FUNCTION_BLOCK KnownExamplesTest EXTENDS TcUnit_Zeugwerk.FB_TestSuite

example01();
example02();
example03();
example04();
example05();
example06();
example07();
example08();
example09();
example10();
example11();
example12();
example13();
example14();
example15();
example16();
example17();
example18();
example19();
example20();
example21();
example22();
example23();
example24();
example25();
example26();
example27();
example28();
example29();
example30();
example31();
example32();
example33();
example34();
example35();
example36();
example37();

METHOD example01
VAR_INST
  otg : Struckig.Otg(0.005, 3) := (
  
    Synchronization := SynchronizationType.None,        
    MaxVelocity :=         [ 1.0, 1.0, 1.0 ],
    MaxAcceleration :=     [ 1.0, 1.0, 1.0 ],
    MaxJerk :=             [ 1.0, 1.0, 1.0 ],
    CurrentPosition :=     [ 0.0, 0.0, 0.0 ],
    CurrentVelocity :=     [ 0.0, 0.0, 0.0 ],
    CurrentAcceleration := [ 0.0, 0.0, 0.0 ],
    TargetPosition :=      [ 0.0, 0.0, 0.0 ],
    TargetVelocity :=      [ 0.0, 0.0, 0.0 ],
    TargetAcceleration :=  [ 0.0, 0.0, 0.0 ]
  );
  
END_VAR
TEST('Example-01');

otg();
AssertEquals_LREAL(Expected := 0.0,
             Actual := CheckCalculation(otg),
             DELTA := 1E-8,
             Message := '');
 
TEST_FINISHED();
END_METHOD

METHOD example02
VAR_INST
  otg : Struckig.Otg(0.005, 3) := (
  
    Synchronization := SynchronizationType.None,        
    MaxVelocity :=         [ 1.0, 1.0, 1.0 ],
    MaxAcceleration :=     [ 1.0, 1.0, 1.0 ],
    MaxJerk :=             [ 1.0, 1.0, 1.0 ],
    CurrentPosition :=     [ 0.0, 0.0, 0.0 ],
    CurrentVelocity :=     [ 0.0, 0.0, 0.0 ],
    CurrentAcceleration := [ 0.0, 0.0, 0.0 ],
    TargetPosition :=      [ 0.0, 1E-17, -1E-17 ],
    TargetVelocity :=      [ 0.0, 0.0, 0.0 ],
    TargetAcceleration :=  [ 0.0, 0.0, 0.0 ]
  );
    
END_VAR
TEST('Example-02');

otg();
AssertEquals_LREAL(Expected := 1E-18,
             Actual := CheckCalculation(otg),
             Delta := 1E-8,
             Message := '');
 
TEST_FINISHED();
END_METHOD

METHOD example03
VAR_INST
  otg : Struckig.Otg(0.005, 3) := (
  
    Synchronization := SynchronizationType.None,        
    MaxVelocity :=         [ 1.0, 1.0, 1.0 ],
    MaxAcceleration :=     [ 1.0, 1.0, 1.0 ],
    MaxJerk :=             [ 1.0, 1.0, 1.0 ],
    CurrentPosition :=     [ 0.0, 1E-17, -1E-17 ],
    CurrentVelocity :=     [ 0.0, 0.0, 0.0 ],
    CurrentAcceleration := [ 0.0, 0.0, 0.0 ],
    TargetPosition :=      [ 1.0, 1.0, 1.0 ],
    TargetVelocity :=      [ 0.0, 0.0, 0.0 ],
    TargetAcceleration :=  [ 0.0, 0.0, 0.0 ]
  );
  
  
END_VAR
TEST('Example-03');

otg();
AssertEquals_LREAL(Expected := 3.1748021039,
             Actual := CheckCalculation(otg),
             DELTA := 1E-8,
             Message := '');
 
TEST_FINISHED();
END_METHOD

METHOD example04
VAR_INST
  otg : Struckig.Otg(0.005, 3) := (
  
    Synchronization := SynchronizationType.None,        
    MaxVelocity :=         [ 1.0, 1.0, 1.0 ],
    MaxAcceleration :=     [ 1.0, 1.0, 1.0 ],
    MaxJerk :=             [ 2.0, 2.0, 2.0 ],
    CurrentPosition :=     [ 0.0, 0.0, 0.0 ],
    CurrentVelocity :=     [ 0.0, 0.0, 0.0 ],
    CurrentAcceleration := [ 0.0, 0.0, 0.0 ],
    TargetPosition :=      [ 1.0, 1.0, 1.0 ],
    TargetVelocity :=      [ 0.0, 0.0, 0.0 ],
    TargetAcceleration :=  [ 0.0, 0.0, 0.0 ]
  );
  
  
END_VAR
TEST('Example-04');

otg();
AssertEquals_LREAL(Expected := 2.5615528128,
             Actual := CheckCalculation(otg),
             DELTA := 1E-8,
             Message := '');
 
TEST_FINISHED();
END_METHOD

METHOD example05
VAR_INST
  otg : Struckig.Otg(0.005, 3) := (
  
    Synchronization := SynchronizationType.None,        
    MaxVelocity :=         [ 0.6, 0.6, 0.6 ],
    MaxAcceleration :=     [ 1.0, 1.0, 1.0 ],
    MaxJerk :=             [ 2.0, 2.0, 2.0 ],
    CurrentPosition :=     [ 0.0, 0.0, 0.0 ],
    CurrentVelocity :=     [ 0.0, 0.0, 0.0 ],
    CurrentAcceleration := [ 0.0, 0.0, 0.0 ],
    TargetPosition :=      [ 1.0, 1.0, 1.0 ],
    TargetVelocity :=      [ 0.0, 0.0, 0.0 ],
    TargetAcceleration :=  [ 0.0, 0.0, 0.0 ]
  );
  
  
END_VAR
TEST('Example-05');

otg();
AssertEquals_LREAL(Expected := 2.7666666667,
             Actual := CheckCalculation(otg),
             DELTA := 1E-8,
             Message := '');
 
TEST_FINISHED();
END_METHOD

METHOD example06
VAR_INST
  otg : Struckig.Otg(0.005, 3) := (
  
    Synchronization := SynchronizationType.None,        
    MaxVelocity :=         [ 0.4, 0.4, 0.4 ],
    MaxAcceleration :=     [ 1.0, 1.0, 1.0 ],
    MaxJerk :=             [ 2.0, 2.0, 2.0 ],
    CurrentPosition :=     [ 0.0, 0.0, 0.0 ],
    CurrentVelocity :=     [ 0.0, 0.0, 0.0 ],
    CurrentAcceleration := [ 0.0, 0.0, 0.0 ],
    TargetPosition :=      [ 1.0, 1.0, 1.0 ],
    TargetVelocity :=      [ 0.0, 0.0, 0.0 ],
    TargetAcceleration :=  [ 0.0, 0.0, 0.0 ]
  );
  	
END_VAR
TEST('Example-06');

otg();
AssertEquals_LREAL(Expected := 3.394427191,
             Actual := CheckCalculation(otg),
             DELTA := 1E-8,
             Message := '');
 
TEST_FINISHED();
END_METHOD

METHOD example07
VAR_INST
  otg : Struckig.Otg(0.005, 3) := (
  
    Synchronization := SynchronizationType.None,        
    MaxVelocity :=         [ 1.0, 1.0, 1.0 ],
    MaxAcceleration :=     [ 1.0, 1.0, 1.0 ],
    MaxJerk :=             [ 2.0, 2.0, 2.0 ],
    CurrentPosition :=     [ 0.0, 0.0, 0.0 ],
    CurrentVelocity :=     [ 0.3, 0.3, 0.3 ],
    CurrentAcceleration := [ 0.0, 0.0, 0.0 ],
    TargetPosition :=      [ 1.0, 1.0, 1.0 ],
    TargetVelocity :=      [ 0.0, 0.0, 0.0 ],
    TargetAcceleration :=  [ 0.0, 0.0, 0.0 ]
  );
  
  
END_VAR
TEST('Example-07');

otg();
AssertEquals_LREAL(Expected := 2.2319602829,
             Actual := CheckCalculation(otg),
             DELTA := 1E-8,
             Message := '');
 
TEST_FINISHED();
END_METHOD

METHOD example08
VAR_INST
  otg : Struckig.Otg(0.005, 3) := (
  
    Synchronization := SynchronizationType.None,        
    MaxVelocity :=         [ 0.6, 0.6, 0.6 ],
    MaxAcceleration :=     [ 1.0, 1.0, 1.0 ],
    MaxJerk :=             [ 2.0, 2.0, 2.0 ],
    CurrentPosition :=     [ 0.0, 0.0, 0.0 ],
    CurrentVelocity :=     [ 0.3, 0.3, 0.3 ],
    CurrentAcceleration := [ 0.0, 0.0, 0.0 ],
    TargetPosition :=      [ 1.0, 1.0, 1.0 ],
    TargetVelocity :=      [ 0.0, 0.0, 0.0 ],
    TargetAcceleration :=  [ 0.0, 0.0, 0.0 ]
  );
  
  
END_VAR
TEST('Example-08');

otg();
AssertEquals_LREAL(Expected := 2.410315834,
             Actual := CheckCalculation(otg),
             DELTA := 1E-8,
             Message := '');
 
TEST_FINISHED();
END_METHOD

METHOD example09
VAR_INST
  otg : Struckig.Otg(0.005, 3) := (
  
    Synchronization := SynchronizationType.None,        
    MaxVelocity :=         [ 0.6, 0.6, 0.6 ],
    MaxAcceleration :=     [ 1.0, 1.0, 1.0 ],
    MaxJerk :=             [ 2.0, 2.0, 2.0 ],
    CurrentPosition :=     [ 0.0, 0.0, 0.0 ],
    CurrentVelocity :=     [ 0.0, 0.0, 0.0 ],
    CurrentAcceleration := [ 0.0, 0.0, 0.0 ],
    TargetPosition :=      [ -1.0, -1.0, -1.0 ],
    TargetVelocity :=      [ 0.0, 0.0, 0.0 ],
    TargetAcceleration :=  [ 0.0, 0.0, 0.0 ]
  );
  
  
END_VAR
TEST('Example-09');

otg();
AssertEquals_LREAL(Expected := 2.7666666667,
             Actual := CheckCalculation(otg),
             DELTA := 1E-8,
             Message := '');
 
TEST_FINISHED();
END_METHOD

METHOD example10
VAR_INST
  otg : Struckig.Otg(0.005, 3) := (
  
    Synchronization := SynchronizationType.None,        
    MaxVelocity :=         [ 10.0, 10.0, 10.0 ],
    MaxAcceleration :=     [ 10.0, 10.0, 10.0 ],
    MaxJerk :=             [ 2.0, 2.0, 2.0 ],
    CurrentPosition :=     [ 0.0, 0.0, 0.0 ],
    CurrentVelocity :=     [ 0.2, 0.2, 0.2 ],
    CurrentAcceleration := [ 0.0, 0.0, 0.0 ],
    TargetPosition :=      [ -1.0, -1.0, -1.0 ],
    TargetVelocity :=      [ 0.0, 0.0, 0.0 ],
    TargetAcceleration :=  [ 0.0, 0.0, 0.0 ]
  );
  
END_VAR
TEST('Example-10');

otg();
AssertEquals_LREAL(Expected := 2.7338531701,
             Actual := CheckCalculation(otg),
             DELTA := 1E-8,
             Message := '');
 
TEST_FINISHED();
END_METHOD

METHOD example11
VAR_INST
  otg : Struckig.Otg(0.005, 3) := (
  
    Synchronization := SynchronizationType.None,        
    MaxVelocity :=         [ 0.4, 0.4, 0.4 ],
    MaxAcceleration :=     [ 1.0, 1.0, 1.0 ],
    MaxJerk :=             [ 2.0, 2.0, 2.0 ],
    CurrentPosition :=     [ -1.0, -1.0, -1.0 ],
    CurrentVelocity :=     [ 0.2, 0.2, 0.2 ],
    CurrentAcceleration := [ 0.0, 0.0, 0.0 ],
    TargetPosition :=      [ 1.0, 1.0, 1.0 ],
    TargetVelocity :=      [ 0.0, 0.0, 0.0 ],
    TargetAcceleration :=  [ 0.0, 0.0, 0.0 ]
  );
  
  
END_VAR
TEST('Example-11');

otg();
AssertEquals_LREAL(Expected := 5.6053274785,
             Actual := CheckCalculation(otg),
             DELTA := 1E-8,
             Message := '');
 
TEST_FINISHED();
END_METHOD

METHOD example12
VAR_INST
  otg : Struckig.Otg(0.005, 3) := (
  
    Synchronization := SynchronizationType.None,        
    MaxVelocity :=         [ 3.0, 3.0, 3.0 ],
    MaxAcceleration :=     [ 0.5, 0.5, 0.5 ],
    MaxJerk :=             [ 0.2, 0.2, 0.2 ],
    CurrentPosition :=     [ 0.3888899206957 - 10E-14, 0.0, 0.0 ],
    CurrentVelocity :=     [ 0.2231429352410215, 0.0, 0.0 ],
    CurrentAcceleration := [ -0.2987593916455, 0.0, 0.0 ],
    TargetPosition :=      [ 0.5, 0.0, 0.0 ],
    TargetVelocity :=      [ 0.0, 0.0, 0.0 ],
    TargetAcceleration :=  [ 0.0, 0.0, 0.0 ]
  );
  
END_VAR
TEST('Example-12');

otg();
AssertEquals_LREAL(Expected := 1.493796958,
             Actual := CheckCalculation(otg),
             DELTA := 1E-8,
             Message := '');
 
TEST_FINISHED();
END_METHOD

METHOD example13
VAR_INST
  otg : Struckig.Otg(0.005, 3) := (
  
    Synchronization := SynchronizationType.None,        
    MaxVelocity :=         [ 12.9892953062198, 3.74169932927481, 1.42398447457303 ],
    MaxAcceleration :=     [ 4.2162106624246, 10.2906731766853, 2.1869079548297 ],
    MaxJerk :=             [ 8.03496976453435, 0.200684346397485 - 1.0E-14, 0.0848503482861296 ],
    CurrentPosition :=     [ -5.54640573838539, -2.34195463203842, 5.10070661762967 ],
    CurrentVelocity :=     [ 0.824843228617216, -1.03863337183304, -0.749451523227729 ],
    CurrentAcceleration := [ -0.119403564898501, 0.923861820607788, 3.04022341347259 ],
    TargetPosition :=      [ -1.58293112753888, 0.383405919465141, 5.79349604610299 ],
    TargetVelocity :=      [ -1.59453676324393, 0.0, -0.0693173526513803 ],
    TargetAcceleration :=  [ -0.664429703711622, 0.0, 0.0 ]
  );
  
  
END_VAR
TEST('Example-13');

otg();
AssertEquals_LREAL(Expected := 1921.0797627836,
             Actual := CheckCalculation(otg),
             DELTA := 1E-8,
             Message := '');
 
TEST_FINISHED();
END_METHOD

METHOD example14
VAR_INST
  otg : Struckig.Otg(0.005, 3) := (
  
    Synchronization := SynchronizationType.None,        
    MaxVelocity :=         [ 8.65978706670502, 5.94921088330542, 10.7652253566829 ],
    MaxAcceleration :=     [ 3.40137210377608, 4.04166318018487, 10.8617860610581 ],
    MaxJerk :=             [ 10.9542353113865, 3.11056302676629, 0.798055744482636 + 9E-12 ],
    CurrentPosition :=     [ -6.49539540831446, 6.14883133273172, -2.02636240900911 ],
    CurrentVelocity :=     [ -1.14327601654428, 0.00991019970085593, -1.00932863927626 ],
    CurrentAcceleration := [ -1.73501068960131, -0.584885092422228, 0 ],
    TargetPosition :=      [ 4.4676187540058, 2.93367894961155, -0.646008452514058 ],
    TargetVelocity :=      [ -0.544559915133859, 0.298517792372943, 1.6058847848484 ],
    TargetAcceleration :=  [ -1.31832055647831, 0, 0 ]
  );
  
  
END_VAR
TEST('Example-14');

otg();
AssertEquals_LREAL(Expected := 4.6277455678,
             Actual := CheckCalculation(otg),
             DELTA := 1E-8,
             Message := '');
 
TEST_FINISHED();
END_METHOD

METHOD example15
VAR_INST
  otg : Struckig.Otg(0.005, 3) := (
  
    Synchronization := SynchronizationType.TimeSync,        // TODO: there seems to be a bug here, if set to None, the reported duration is <3s
    MaxVelocity :=         [ 7.97399137456765, 2.68591430972239, 9.54987666746364 ],
    MaxAcceleration :=     [ 5.44679859206862, 7.61752909348119, 0.473482772614085 ],
    MaxJerk :=             [ 7.88958080921515, 5.26855927512131, 0.764061581326592 - 1E-14 ],
    CurrentPosition :=     [ 7.06378251402596, -2.4834697862831, -0.843847405371359 ],
    CurrentVelocity :=     [ 0.436985859305842, 0.0708113515655622, -0.751266816040307 ],
    CurrentAcceleration := [ -0.80835350359544, 0, -0.355284934641626 ],
    TargetPosition :=      [ 4.40606827118048, -2.84629921001043, -2.91829890043522 ],
    TargetVelocity :=      [ 0.555084596169823, 0, -1.24631524923535 ],
    TargetAcceleration :=  [ 0.463000173872542, 0, 0 ]
  );
  
  
END_VAR
TEST('Example-15');

otg();
AssertEquals_LREAL(Expected := 8.8739464323,
             Actual := CheckCalculation(otg),
             DELTA := 1E-8,
             Message := '');
 
TEST_FINISHED();
END_METHOD

METHOD example16
VAR_INST
  otg : Struckig.Otg(0.005, 3) := (
  
    Synchronization := SynchronizationType.None,        
    MaxVelocity :=         [ 0.1241065584614779, 1, 1 ],
    MaxAcceleration :=     [ 1.808598147153279, 1, 1 ],
    MaxJerk :=             [ 2.516849090900998 - 3E-15, 1, 1 ],
    CurrentPosition :=     [ -7.962737259350095, 0, 0 ],
    CurrentVelocity :=     [ -0.8844863500141733, 0, 0 ],
    CurrentAcceleration := [ 2.252932547031004, 0, 0 ],
    TargetPosition :=      [ -3.547368989678775, 0, 0 ],
    TargetVelocity :=      [ 0, 0, 0 ],
    TargetAcceleration :=  [ 0.217242176687843, 0, 0 ]
  );
  
  
END_VAR
TEST('Example-16');

otg();
AssertEquals_LREAL(Expected := 38.3409477609,
             Actual := CheckCalculation(otg),
             DELTA := 1E-8,
             Message := '');
 
TEST_FINISHED();
END_METHOD

METHOD example17
VAR_INST
  otg : Struckig.Otg(0.005, 3) := (
  
    Synchronization := SynchronizationType.None,    
    MaxVelocity :=         [ 1.863775561344568, 0.4357836109021987, 6.260907804906162 ],
    MaxAcceleration :=     [ 9.49223908896113, 9.002562577262177, 1.119142029086944 ],
    MaxJerk :=             [ 8.689575453772798, 0.09322235504216797, 0.1594452521517275 + 3E-15 ],
    CurrentPosition :=     [ -4.180150148354134, 1.030371049895473, -2.660154279239869 ],
    CurrentVelocity :=     [ 1.673805463302308, -1.435796222257198, 0.9711306630275642 ],
    CurrentAcceleration := [ 1.412175048500792, 1.892262449040863, -1.128847905860926 ],
    TargetPosition :=      [ 2.079913937916431, 1.839862681333277, 2.341421542126605 ],
    TargetVelocity :=      [ 0.7537566830764975, 0, 0.02507782261105568 ],
    TargetAcceleration :=  [ -0.8610296259045267, -0.07876324073516261, 0 ]
  );
  
  
END_VAR
TEST('Example-17');

otg();
AssertEquals_LREAL(Expected := 1135.0135089249,
             Actual := CheckCalculation(otg),
             DELTA := 1E-8,
             Message := '');
 
TEST_FINISHED();
END_METHOD

METHOD example18
VAR_INST
  otg : Struckig.Otg(0.005, 3) := (
  
    Synchronization := SynchronizationType.None,
    MaxVelocity :=         [ 6.144314006624488, 2.93258338415229, 0.1820021269527196 ],
    MaxAcceleration :=     [ 5.199401036221791, 1.848176490768948, 11.11168017805234 ],
    MaxJerk :=             [ 9.940940357283978, 10.46997753899755, 0.08166297169205029 ],
    CurrentPosition :=     [ -4.490717417930574, 3.467236624628543, -0.7545929089757601 ],
    CurrentVelocity :=     [ 0.1839756723363622, -0.4356283320280516, 0.7490399525818022 ],
    CurrentAcceleration := [ -1.057769973808928, 0, -2.368645439140517 ],
    TargetPosition :=      [ -4.928244836531066, -4.821780824003112, -8.20567952461017 ],
    TargetVelocity :=      [ 0.1097319156272965, -0.9272874846270881, 0 ],
    TargetAcceleration :=  [ 0.03089046366221739, -0.9744054582899561, 0 ]
  );
  
  
END_VAR
TEST('Example-18');

otg();
AssertEquals_LREAL(Expected := 7295.4375633935,
             Actual := CheckCalculation(otg),
             DELTA := 1E-8,
             Message := '');
 
TEST_FINISHED();
END_METHOD

METHOD example19
VAR_INST
  otg : Struckig.Otg(0.005, 3) := (
  
    Synchronization := SynchronizationType.None,
    MaxVelocity :=         [ 1, 1, 1 ],
    MaxAcceleration :=     [ 7, 7, 7 ],
    MaxJerk :=             [ 1000, 1000, 1000 ],
    CurrentPosition :=     [ 0.01073568005271233, -0.7002627264230739, 0 ],
    CurrentVelocity :=     [ 0.05656281587106524, 1.011281770884991, 0 ],
    CurrentAcceleration := [ -5.348847133445708, -3.400994300842285, 0 ],
    TargetPosition :=      [ 0.0698, 0.6283, 0 ],
    TargetVelocity :=      [ 0, 0, 0 ],
    TargetAcceleration :=  [ 0, 0, 0 ]
  );
  
  
END_VAR
TEST('Example-19');

otg();
AssertEquals_LREAL(Expected := 1.403613276,
             Actual := CheckCalculation(otg),
             DELTA := 1E-3,
             Message := '');
 
TEST_FINISHED();
END_METHOD

METHOD example20
VAR_INST
  otg : Struckig.Otg(0.005, 3) := (
  
    Synchronization := SynchronizationType.None,
    MaxVelocity :=         [ 1, 1, 1 ],
    MaxAcceleration :=     [ 0.5, 0.5, 0.5 ],
    MaxJerk :=             [ 1, 1, 1 ],
    CurrentPosition :=     [ 0.0001215, 0, 0 ],
    CurrentVelocity :=     [ 0.00405, 0, 0 ],
    CurrentAcceleration := [ 0.09, 0, 0 ],
    TargetPosition :=      [ 0.1421083333333333087, 0, 0 ],
    TargetVelocity :=      [ 0.37, 0, 0 ],
    TargetAcceleration :=  [ 0.5, 0, 0 ]
  );
  
  
END_VAR
TEST('Example-20');

otg();
AssertEquals_LREAL(Expected := 0.9,
             Actual := CheckCalculation(otg),
             DELTA := 1E-8,
             Message := '');
 
TEST_FINISHED();
END_METHOD

METHOD example21
VAR_INST
  otg : Struckig.Otg(0.005, 3) := (
  
    Synchronization := SynchronizationType.None,
    MaxVelocity :=         [ 1800, 18000, 180000 ],
    MaxAcceleration :=     [ 20000, 200000, 2000000 ],
    MaxJerk :=             [ 200000, 2000000, 20000000 ],
    CurrentPosition :=     [ 0, 0, 0 ],
    CurrentVelocity :=     [ 0, 0, 0 ],
    CurrentAcceleration := [ 0, 0, 0 ],
    TargetPosition :=      [ 400, 4000, 40000 ],
    TargetVelocity :=      [ 0, 0, 0 ],
    TargetAcceleration :=  [ 0, 0, 0 ]
  );
  
  
END_VAR
TEST('Example-21');

otg();
AssertEquals_LREAL(Expected := 0.4119588818,
             Actual := CheckCalculation(otg),
             DELTA := 1E-8,
             Message := '');
 
TEST_FINISHED();
END_METHOD

METHOD example22
VAR_INST
  otg : Struckig.Otg(0.005, 3) := (
  
    Synchronization := SynchronizationType.None,
    MaxVelocity :=         [ 0.8500000000000001, 0.8500000000000001, 0.8500000000000001 ],
    MaxAcceleration :=     [ 4.25, 4.25, 4.25 ],
    MaxJerk :=             [ 85.00000000000001, 85.00000000000001, 85.00000000000001 ],
    CurrentPosition :=     [ -0.05598571695553641, -0.534847776106059, 0.0978130731424748 ],
    CurrentVelocity :=     [ -0.03425673149926184, -0.8169926404190487, -0.004506245841081729 ],
    CurrentAcceleration := [ -2.720000000000001, 1.440254448401435, 0 ],
    TargetPosition :=      [ -0.0534691276550293, -0.6224863891601563, 0.09690575408935546 ],
    TargetVelocity :=      [ 0, 0, 0 ],
    TargetAcceleration :=  [ 0, 0, 0 ]
  );
  
  
END_VAR
TEST('Example-22');

otg();
AssertEquals_LREAL(Expected := 0.2281604414,
             Actual := CheckCalculation(otg),
             DELTA := 1E-8,
             Message := '');
 
TEST_FINISHED();
END_METHOD

METHOD example23
VAR_INST
  otg : Struckig.Otg(0.005, 3) := (
  
    Synchronization := SynchronizationType.None,
    MaxVelocity :=         [ 1.0, 1.0, 10.01369296498101 ],
    MaxAcceleration :=     [ 1.0, 1.0, 14.72621077848741 ],
    MaxJerk :=             [ 1.0, 1.0, 7.770133554060553 ],
    CurrentPosition :=     [ 0.0, 0.0, 0.3736320740840176 ],
    CurrentVelocity :=     [ 0.0, 0.0, -0.60486324450823 ],
    CurrentAcceleration := [ 0.0, 0.0, -0.4953501898933239 ],
    TargetPosition :=      [ 0.0, 0.0, 0.233562911156468 ],
    TargetVelocity :=      [ 0, 0, 0 ],
    TargetAcceleration :=  [ 0, 0, 0 ],
    MinVelocity :=         [ -1.0, -1.0, -1.94898305867544],
    MinAcceleration :=     [ -1.0, -1.0, -0.6829625196960336]
  );
  
  
END_VAR
TEST('Example-23');

otg();
AssertEquals_LREAL(Expected := 1.08732372,
             Actual := CheckCalculation(otg),
             DELTA := 1E-8,
             Message := '');
 
TEST_FINISHED();
END_METHOD

METHOD example24
VAR_INST
  otg : Struckig.Otg(0.005, 3) := (
    MaxVelocity :=         [ 14.64378197125325, 3.0, 3.0 ],
    MaxAcceleration :=     [ 0.4552736879216988, 2.5, 2.5 ],
    MaxJerk :=             [ 12.15045820314999, 2.2, 2.2 ],
    CurrentPosition :=     [ -0.01919986582215404, 0.0, 0.0 ],
    CurrentVelocity :=     [ -0.3858205249368821, 0.0, 0.0 ],
    CurrentAcceleration := [ 0.1889847091893647, 0.0, 0.0 ],
    TargetPosition :=      [ 1.297187158009963, 0.0, 0.0 ],
    TargetVelocity :=      [ 1.160424379732321, 0.0, 0.0 ],
    TargetAcceleration :=  [ 0.4552736879206988, 0.0, 0.0 ],
    MinVelocity :=         [ -1.0, -1.0, -1.94898305867544],
    MinAcceleration :=     [ -1.0, -1.0, -0.6829625196960336],
    MinDuration := 3.408914
  );
  
  
END_VAR
TEST('Example-24');

otg();
AssertEquals_LREAL(Expected := 3.408914,
             Actual := CheckCalculation(otg),
             DELTA := 1E-8,
             Message := '');
 
TEST_FINISHED();
END_METHOD

METHOD example25
VAR_INST
  otg : Struckig.Otg(0.004, 3) := (
    MaxVelocity :=         [ 0.25, 0.25, 0.25 ],
    MaxAcceleration :=     [ 2.5, 2.5, 2.5 ],
    MaxJerk :=             [ 62.5, 62.5, 62.5 ],
    CurrentPosition :=     [ 0.2473592757796861, 0.2921606775204735, 0.7758663276711127 ],
    CurrentVelocity :=     [ -0.2426115138900957, 0.2200706500820608, -0.01891492763905089 ],
    CurrentAcceleration := [ 0.01877538437863763, -0.6573642866096158, 0.5 ],
    TargetPosition :=      [ 0.2308075286416321, 0.3066442218484541, 0.7733155040940536 ],
    TargetVelocity :=      [ 0.0, 0.0, 0.0 ],
    TargetAcceleration :=  [ 0.0, 0.0, 0.0 ],
    Discretization := DiscretizationType.Discrete
  );
  
  
END_VAR
TEST('Example-25');

otg();
AssertEquals_LREAL(Expected := 0.14,
             Actual := CheckCalculation(otg),
             DELTA := 1E-8,
             Message := '');
 
TEST_FINISHED();
END_METHOD

METHOD example26
VAR_INST
  otg : Struckig.Otg(0.004, 3) := (
    MaxVelocity :=         [ 1, 1 ,1 ],
    MaxAcceleration :=     [ 10, 10, 10 ],
    MaxJerk :=             [ 100 + 1E-14, 100 + 1E-14, 100 + 1E-14 ],
    CurrentPosition :=     [ 0.02853333333333339, 0.0285, 0.0285 ],
    CurrentVelocity :=     [ 0.6800000000000006, 0.68, 0.68 ],
    CurrentAcceleration := [ 7.999999999999993, 8.0, 8.0 ],
    TargetPosition :=      [ 0, 0, 0 ],
    TargetVelocity :=      [ 0.0, 0.0, 0.0 ],
    TargetAcceleration :=  [ 0.0, 0.0, 0.0 ],
    Discretization := DiscretizationType.Discrete
  );
  
  
END_VAR
TEST('Example-26');

otg();
AssertEquals_LREAL(Expected := 0.58,
             Actual := CheckCalculation(otg),
             DELTA := 1E-8,
             Message := '');
 
TEST_FINISHED();
END_METHOD

METHOD example27
VAR_INST
  otg : Struckig.Otg(0.004, 3) := (
    MaxVelocity :=         [ 6.457718232379019, 5.410520681182422, 7.155849933176751 ],
    MaxAcceleration :=     [ 26.89552377323262, 22.5322006432468, 29.81022362406315 ],
    MaxJerk :=             [ 224.2224490037115, 187.8497873921497, 248.4650723139127 ],
    CurrentPosition :=     [ 0.5289912019692077, -0.2461593579591288, -0.2728396804501142 ],
    CurrentVelocity :=     [ 0.0287779218983349, -0.005980397028399779, 0.04763314105835294 ],
    CurrentAcceleration := [ -1.374657509445135, 0.2564786317266955, -2.497210506808601 ],
    TargetPosition :=      [ 0, 0, 0 ],
    TargetVelocity :=      [ 0.0, 0.0, 0.0 ],
    TargetAcceleration :=  [ 0.0, 0.0, 0.0 ],
    Discretization := DiscretizationType.Discrete,
    ControlInterface := ControlInterfaceType.Velocity
  );
  
  
END_VAR
TEST('Example-27');

otg();
AssertEquals_LREAL(Expected :=0.024,
             Actual := CheckCalculation(otg),
             DELTA := 1E-8,
             Message := '');
 
TEST_FINISHED();
END_METHOD

METHOD example28
VAR_INST
  otg : Struckig.Otg(0.004, 3) := (
    MaxVelocity :=         [ 10.0, 10.0, 10.0 ],
    MaxAcceleration :=     [ 10.0, 10.0, 10.0 ],
    MaxJerk :=             [ 224.2224490037115, 187.8497873921497, 10.0 ],
    CurrentPosition :=     [ 0.0, 0.0, 0.0 ],
    CurrentVelocity :=     [ 0.1119477497536703, -0.005706738140158095, 0.0 ],
    CurrentAcceleration := [ -2.943871184141059, 0.1638588832925878, 0.0 ],
    TargetPosition :=      [ 0, 0, 0 ],
    TargetVelocity :=      [ 0.0, 0.0, 0.0 ],
    TargetAcceleration :=  [ 0.0, 0.0, 0.0 ],
    Discretization := DiscretizationType.Continuous,
    ControlInterface := ControlInterfaceType.Velocity
  );
END_VAR
TEST('Example-28');

otg();
AssertEquals_LREAL(Expected := 0.0352632,
             Actual := CheckCalculation(otg),
             DELTA := 1E-7,
             Message := '');
 
TEST_FINISHED();
END_METHOD

METHOD example29
VAR_INST
  otg : Struckig.Otg(0.004, 6) := (
    CurrentPosition := [0.5, -0.7, -0.7, -1.5, -0, -0.2],
    CurrentVelocity := [2.689534009085704E-06, -2.689534009088848E-06, -2.689534009086246E-06, -2.689534009088414E-06, 2.689534009087655E-06, -2.689534009089241E-06],
    CurrentAcceleration := [-0.001639979880695402, 0.001639979880696266, 0.001639979880695815, 0.00163997988069603, -0.00163997988069612],
    TargetPosition := [1.5, -0.7, -0.7, -1.5, 0, -0.2],
    TargetVelocity := [0, 0, 0, 0, 0, 0 ],
    TargetAcceleration := [0, 0, 0, 0, 0, 0],
    MaxVelocity := [0.5, 0.5, 0.5, 0.5, 0.5, 0.5],
    MaxAcceleration := [0.5, 0.5, 0.5, 0.5, 0.5, 0.5],
    MaxJerk := [0.5, 0.5, 0.5, 0.5, 0.5, 0.5]
  );
END_VAR
TEST('Example-29');

otg();
AssertEquals_LREAL(Expected := 4.0032799558,
             Actual := CheckCalculation(otg),
             DELTA := 1E-7,
             Message := '');
 
TEST_FINISHED();
END_METHOD

METHOD example30
VAR_INST
  otg : Struckig.Otg(0.004, 3) := (
    CurrentPosition := [0.0, 0.0, 0.0],
    CurrentVelocity := [1.0, 0.0, 0.0],
    CurrentAcceleration := [0.0, 0.0, 0.0],
    TargetPosition := [0.0, 0.0, 0.0],
    TargetVelocity := [1.0, 0.0, 1.0],
    TargetAcceleration := [0.0, 0.0, 0.0],
    MaxVelocity := [1.0, 1.0, 1.0],
    MaxAcceleration := [1.0, 1.0, 1.0],
    MaxJerk := [1.0, 1.0, 1.0],
    ControlInterface := ControlInterfaceType.Velocity
  );
END_VAR
TEST('Example-30');

otg();
AssertEquals_LREAL(Expected := 2.0,
             Actual := CheckCalculation(otg),
             DELTA := 1E-7,
             Message := '');
 
TEST_FINISHED();
END_METHOD

METHOD example31
VAR_INST
  otg : Struckig.Otg(0.004, 3) := (
    CurrentPosition := [-0.54516231864478149, -1.4206629551476477, 0.32727720821160067],
    CurrentVelocity := [6.1348323207600686, -0.0040477518609957240, 0.0088178054233364854],
    CurrentAcceleration := [0.0000000000000000, 0.19725113486681556, -0.23382835447542066],
    TargetVelocity := [6.1348323207600686, 0.014259490365703332, -0.012798219033181931],
    TargetAcceleration := [0.0, 0.0, 0.0],
    MaxVelocity := [6.4577182323790190, 5.4105206811824216, 7.1558499331767509],
    MaxAcceleration := [26.895523773232618, 22.532200643246796, 29.810223624063148],
    MaxJerk := [224.22244900371152, 187.84978739214969, 248.46507231391274],
    ControlInterface := ControlInterfaceType.Velocity
  );
END_VAR
TEST('Example-31');

otg();
AssertEquals_LREAL(Expected := 0.0187497625,
             Actual := CheckCalculation(otg),
             DELTA := 1E-7,
             Message := '');
 
TEST_FINISHED();
END_METHOD

METHOD example32
VAR_INST
  otg : Struckig.Otg(0.004, 3) := (
    CurrentPosition := [-1.2563817016634644, -0.51079124473334669, 2.4607439315667303],
    CurrentVelocity := [3.4194572623820010, 5.7548168684509085, -1.5675191369761612],
    CurrentAcceleration := [27.722541632719086, -1.7945991957745204, -22.971380686605098],
    TargetVelocity := [5.1559110036108979, 5.5636136585722848, -3.6173923596604807],
    TargetAcceleration := [0.0, 0.0, 0.0],
    MaxVelocity := [9.5993108859688121, 9.4247779607693793, 17.453292519943297],
    MaxAcceleration := [39.985493163190093, 39.618974020271281, 72.710416638083771],
    MaxJerk := [333.30552725335713, 330.26865435488696, 606.01322287747109],
    ControlInterface := ControlInterfaceType.Velocity
  );
END_VAR
TEST('Example-32');

otg();
AssertEquals_LREAL(Expected := 0.1030382161,
             Actual := CheckCalculation(otg),
             DELTA := 1E-7,
             Message := '');
 
TEST_FINISHED();
END_METHOD

METHOD example33
VAR_INST
  otg : Struckig.Otg(0.004, 3) := (
    CurrentPosition := [0, 0, 0],
    CurrentVelocity := [0, -0.0577630321017372216, 0],
    CurrentAcceleration := [0, -1.9198621771937627, 0],
    TargetPosition := [0, 0, 0],
    TargetVelocity := [0, -0.1, 0],
    TargetAcceleration := [0.0, 0.0, 0.0],
    MaxVelocity := [5.23, 3.926990816987241394, 3.92],
    MaxAcceleration := [4.36, 4.363323129985824, 4.36],
    MaxJerk := [43.63, 43.633231299858238116, 43.63],
    ControlInterface := ControlInterfaceType.Velocity,
    Discretization := DiscretizationType.Discrete
  );
END_VAR
TEST('Example-33');

otg();
AssertEquals_LREAL(Expected := 0.044,
             Actual := CheckCalculation(otg),
             DELTA := 1E-7,
             Message := '');
 
TEST_FINISHED();
END_METHOD

METHOD example34
VAR_INST
  otg : Struckig.Otg(0.01, 1) := (
    CurrentPosition := [0],
    CurrentVelocity := [1],
    CurrentAcceleration := [-2],
    TargetPosition := [1],
    TargetVelocity := [0.5],
    TargetAcceleration := [0.0],
    MaxVelocity := [0.8],
    MaxAcceleration := [2],
    MaxJerk := [5]
  );
END_VAR
TEST('Example-34');

otg();
AssertEquals_LREAL(Expected := 1.6041105549250121,
             Actual := CheckCalculation(otg),
             DELTA := 1E-7,
             Message := '');
 
TEST_FINISHED();
END_METHOD

METHOD example35
VAR_INST
  otg : Struckig.Otg(0.004, 6) := (
    CurrentPosition := [0.1720894642466409, 3.62255615705579, 1.675754445058354, 2.181127634157466, 0.7829547024446563, 0],
    CurrentVelocity := [0, -0.06422550797049381, -0.006910864193129071, 0.1207111377965507, 0, 0],
    CurrentAcceleration := [0, 0, 0, -0.3999999999978001, 0, 0],
    TargetPosition := [0.1703441349946466, 3.587689540855463, 1.671344092861895, 2.271916653384632, 0.7826056365942573, -0.003141592653589793],
    TargetVelocity := [0, -0.06423623454575711, -0.007006078877926925, 0.1187909578397501, 0, 0],
    TargetAcceleration := [0, 0, 0, 0, 0, 0],
    MaxVelocity := [0.06981316999999999, 0.06423623454575711, 0.007006078877926925, 0.1187909578397501, 6.981317008, 34.90658504],
    MaxAcceleration := [0.034906585, 0.261799388, 0.043633231, 0.4, 4.01425728, 34.90658504],
    MaxJerk := [100, 100, 100, 100, 100, 100]
  );
END_VAR
TEST('Example-35');

otg();
AssertEquals_LREAL(Expected := 0.76427371316291570,
             Actual := CheckCalculation(otg),
             DELTA := 1E-3,
             Message := '');
 
TEST_FINISHED();
END_METHOD

METHOD example36
VAR_INST
  otg : Struckig.Otg(0.004, 6) := (
    CurrentPosition := [0.1174161453909641,-0.4222080077114712,0.3003863125814782,2.960444926889819,-0.005791262234199017,-2.364847659719411],
    CurrentVelocity := [-3.662950284795513E-09,-5.585273134233322E-09,0.01325125623820627,1.800912308381978E-08,-1.307199431356758E-09,-1.908875705031016E-08],
    CurrentAcceleration := [1.350015487635199E-07,2.058506025917496E-07,-0.4883877683641483,-6.637435179724953E-07,4.81780898060446E-08,7.035344641338199E-07],
    TargetPosition := [0.117416145324707,-0.4222080078125,0.3006260070800781,2.960444927215576,-0.00579126225784421,-2.364847660064697],
    TargetVelocity := [0.0, 0.0, 0.0, 0.0, 0.0, 0.0],
    TargetAcceleration := [0, 0, 0, 0, 0, 0],
    MaxVelocity := [0.002,0.002,0.002,0.003141592629253865,0.003141592629253865,0.003141592629253865],
    MaxAcceleration := [0.01,0.01,0.01,0.01570796314626932,0.01570796314626932,0.01570796314626932],
    MaxJerk := [ 0.18,0.18,0.18,1.570796314626932,1.570796314626932,1.570796314626932],
    Discretization := DiscretizationType.Discrete
  );
END_VAR
TEST('Example-36');

otg();
AssertEquals_LREAL(Expected := 11198.436000000000,
             Actual := CheckCalculation(otg),
             DELTA := 1E-7,
             Message := '');
 
TEST_FINISHED();
END_METHOD

METHOD example37
VAR_INST
  otg : Struckig.Otg(0.004, 3) := (
    CurrentPosition := [-19.93333333333424, -0.4983333333333563, 0],
    CurrentVelocity := [10, 0.25, 0],
    CurrentAcceleration := [0, 0, 0],
    TargetPosition := [20, 0.5, 0.2],
    TargetVelocity := [10, 0.25, 0],
    TargetAcceleration := [0, 0, 0],
    MaxVelocity := [10, 10, 10],
    MaxAcceleration := [15, 15, 15],
    MaxJerk := [ 15, 5, 2],
    ControlInterface := ControlInterfaceType.Position,
    Discretization := DiscretizationType.Continuous
  );
  NewPosition, NewVelocity, NewAcceleration, NewJerk : ARRAY[0..ParameterList.MaxDoFs] OF LREAL; // Current state   
  NewSection : INT; 
END_VAR
TEST('Example-37');

otg();
AssertEquals_LREAL(Expected := 3.99333,
             Actual := CheckCalculation(otg),
             DELTA := 1E-5,
             Message := '');
             
otg.AtTime(otg.Duration / 2, ADR(NewPosition), ADR(NewVelocity), ADR(NewAcceleration), ADR(NewJerk), ADR(newSection));
AssertEquals_LREAL(NewPosition[0], 0.033333, 1E-5, '');
AssertEquals_LREAL(NewPosition[1], 0.000833, 1E-5, '');


TEST_FINISHED();
END_METHOD

END_FUNCTION_BLOCK

(* stored: Version 1.1.0.1
   POU KnownExamplesTest: Id {892cc348-6b4c-467a-8c49-6bb12eacf8cd}, SpecialFunc None
   Method example01: Id {e63245db-0c87-42fd-8c9c-5b8ef1846274}
   Method example02: Id {3d024e2f-045e-41d5-afe1-10b2f9dc1698}
   Method example03: Id {c4fb8de0-0810-4b7f-89b7-5d18b1207555}
   Method example04: Id {ecd2ca2f-26a8-4bc0-8f82-360135b2e964}
   Method example05: Id {9a23d7f8-b1dc-4571-8f89-9113608544cf}
   Method example06: Id {9538c878-3ff7-4a42-be69-b82162ad302a}
   Method example07: Id {5d21e693-52b1-4a27-b006-a796cc02d372}
   Method example08: Id {63af5e8a-3ae8-470d-86d7-ef161f3ee77a}
   Method example09: Id {0bba80a6-44ca-4252-acc1-bff433e54793}
   Method example10: Id {429e6937-b1d8-4827-8e66-784a4adb2276}
   Method example11: Id {1e352ae4-7bde-4dd2-a814-185a3be9d037}
   Method example12: Id {0c23ba69-6e49-4902-b866-e3838ab35036}
   Method example13: Id {4c2316f6-1de4-4e19-84c4-ea5a6e1687a5}
   Method example14: Id {47840f6e-c938-48f4-bd1d-5caf30f0b4f6}
   Method example15: Id {90fcdf7e-96a6-43f5-bb79-bce3da217a5b}
   Method example16: Id {16a12324-dfbf-4dae-b099-7a5fcc7de151}
   Method example17: Id {ed9b9e5f-7e2f-4410-bf5b-c0dcca3365ee}
   Method example18: Id {2e6c6a48-90d6-425a-ae57-013d63da4fa1}
   Method example19: Id {86ea15a9-bcc7-4c6c-9c52-2686c5495108}
   Method example20: Id {43d3b3f8-bc82-46c0-9aaa-3c876692e06d}
   Method example21: Id {4ad6cce6-8abe-4583-9a30-738f6d405c8e}
   Method example22: Id {4e3ac0f8-cb9f-4fc8-8d40-78c182460065}
   Method example23: Id {8284e48a-9de8-4315-ac04-9a5fe99c460f}
   Method example24: Id {9bdbf18b-8936-4e4b-9ec5-c8b865228622}
   Method example25: Id {00502c12-c4a7-4387-ad3e-5f69878ff72f}
   Method example26: Id {9d52831f-502e-43e5-ad64-72c3d722f78f}
   Method example27: Id {ccc2cdd0-f683-46d4-8ff5-97bafeee7c04}
   Method example28: Id {c48de666-40fb-4f5c-ba77-31f9be3f1f84}
   Method example29: Id {72f060a7-02f9-44b4-840f-b5c4060b1533}
   Method example30: Id {3fede239-06fe-4709-b2c3-430b2caeee89}
   Method example31: Id {2600698e-c9a2-4a83-86cb-ea07e4bbb42a}
   Method example32: Id {b3457ed3-4b32-4da5-80c9-6838ee359551}
   Method example33: Id {68cceb00-3949-4b80-9f97-16b905bba6e5}
   Method example34: Id {2e155773-1620-4e87-8112-8f35ede17200}
   Method example35: Id {40b97033-fdd1-4031-96bb-de1ea46c05fb}
   Method example36: Id {fa162e63-7481-449c-b111-b6324ea37642}
   Method example37: Id {d2aa66df-9473-48fe-abac-70e8722de314} *)
